// TIA Portal V21 export
DATA_BLOCK "DATALOG TRIGGER BLOCK_DB"   // DB310
// stored: InstanceOfName DATALOG TRIGGER BLOCK, InstanceOfType FB
"DATALOG TRIGGER BLOCK"
   // VAR_INPUT
   //    "SET TIME" : Int;
   //    RESET : Bool;
   //    INPUT : Bool;
   // END_VAR
   // VAR_OUTPUT
   //    "PRESENT VALUE OF TIME" : Int;
   //    SEC : Int;
   //    DONE : Bool;
   //    "TRIGGER BIT" : Bool;
   //    "ALARM BIT" : Bool;
   // END_VAR
   // VAR
   //    "TIMER 1" { S7_SetPoint := 'True'} : IEC_TIMER;
   // END_VAR
   // VAR RETAIN
   //    "COUNTER1 0" { S7_SetPoint := 'True'} : IEC_COUNTER;
   //    "COUNTER1 1" { S7_SetPoint := 'True'} : IEC_COUNTER;
   //    TPULSE { S7_SetPoint := 'True'} : IEC_TIMER;
   // END_VAR
BEGIN
END_DATA_BLOCK
